SUBAPPLICATION Uebung_009a (* RampLimitFS *)
  (* Standard: 61499-2; Description: Copyright (c) 2023 Meisterschulen am Ostbahnhof This program and the accompanying materials are made available under the terms of the Eclipse Public License 2.0 which is available at https://www.eclipse.org/legal/epl-2.0/ SPDX-License-Identifier: EPL-2.0 *)
  (* Version 1.0, 2023-10-23, Franz Höpfinger, Meisterschulen am Ostbahnhof *)
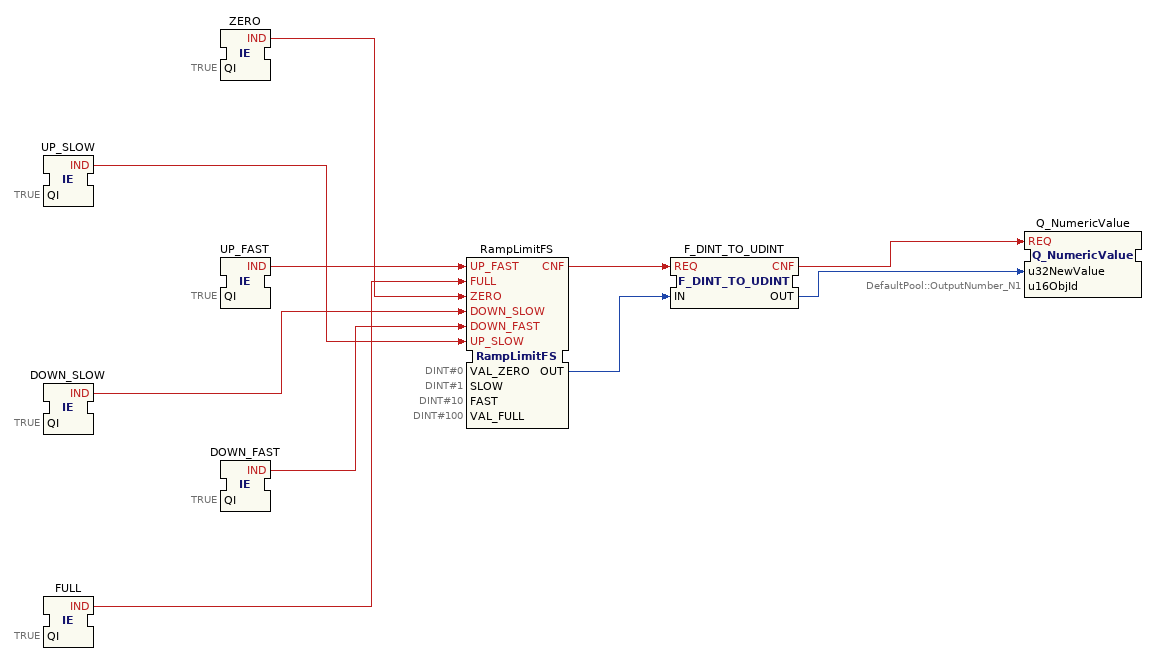
  FBS
    Q_NumericValue : Q_NumericValue(u16ObjId := DefaultPool::OutputNumber_N1);
    UP_FAST : IE(QI := TRUE);
    DOWN_SLOW : IE(QI := TRUE);
    F_DINT_TO_UDINT : F_DINT_TO_UDINT;
    ZERO : IE(QI := TRUE);
    DOWN_FAST : IE(QI := TRUE);
    UP_SLOW : IE(QI := TRUE);
    RampLimitFS : signalprocessing::RampLimitFS(VAL_ZERO := DINT#0, SLOW := DINT#1, FAST := DINT#10, VAL_FULL := DINT#100);
    FULL : IE(QI := TRUE);
  END_FBS
  EVENT_CONNECTIONS
    UP_FAST.IND TO RampLimitFS.UP_FAST;
    FULL.IND TO RampLimitFS.FULL;
    RampLimitFS.CNF TO F_DINT_TO_UDINT.REQ;
    ZERO.IND TO RampLimitFS.ZERO;
    DOWN_SLOW.IND TO RampLimitFS.DOWN_SLOW;
    DOWN_FAST.IND TO RampLimitFS.DOWN_FAST;
    UP_SLOW.IND TO RampLimitFS.UP_SLOW;
    F_DINT_TO_UDINT.CNF TO Q_NumericValue.REQ;
  END_CONNECTIONS
  DATA_CONNECTIONS
    RampLimitFS.OUT TO F_DINT_TO_UDINT.IN;
    F_DINT_TO_UDINT.OUT TO Q_NumericValue.u32NewValue;
  END_CONNECTIONS
END_SUBAPPLICATION
